TYPE CamOut_Statuses_typ EXTENDS MultiAxis_Status_typ :
STRUCT
END_STRUCT
END_TYPE

(* stored: Version 1.1.0.1, ProductVersion 3.1.4024.3
   DUT CamOut_Statuses_typ: Id {1db08190-4fed-09c1-0094-c9708bf8ac51} *)
